// TIA Portal project "function block1" (V16)

(* hardware
DEVICE "S7-1200 station_1"  S7-1200 Station
   slot 0: "Rack_0"  S7-1200 Rack  Rack  V1.0
   slot 1: "PLC_1"  CPU 1214C DC/DC/DC  6ES7 214-1AG40-0XB0  V4.4
   slot 2: "AI 4x13BIT/AQ 2x14BIT_1"  6ES7 234-4HE32-0XB0  V2.1
   slot 101: "CP 1243-7 LTE"  CP 1243-7 LTE  6GK7 243-7KX30-0XE0  V3.2
      slot 0: "Telecontrol server"  Partner
      slot 0: "Inter-station communication"  Partner
   slot 102: "RF120C_1"  RF120C  6GT2 002-0LA00  V1.0
   slot 103: "CM 1243-5"  CM 1243-5  6GK7 243-5DX30-0XE0  V1.3
*)

// ===== PLC "PLC_1"  CPU 1214C DC/DC/DC =====

VAR_GLOBAL   // PLC tag table "Default tag table"
   "switch" AT %M0.0 : Bool;
   "out" AT %M0.1 : Bool;
   "estop" AT %M0.2 : Bool;
   "esnotification" AT %M0.3 : Bool;
   "esalarm" AT %M0.4 : Bool;
   "alarmreset" AT %M0.5 : Bool;
   "alarmsilent" AT %M0.6 : Bool;
END_VAR

DATA_BLOCK "scl_DB"   // DB1
{ S7_Optimized_Access := 'TRUE' }
VERSION : 0.1
// stored: InstanceOfName scl
"scl"
BEGIN
END_DATA_BLOCK

FUNCTION_BLOCK "scl"   // FB1, SCL
{ S7_Optimized_Access := 'TRUE' }
VERSION : 0.1
   VAR
      almset : Bool;
   END_VAR
BEGIN
   IF "estop" AND NOT #almset THEN
       "esalarm" := 1; // Statement section IF
       "esnotification" :=1;
       #almset := 1;
   END_IF;
   IF "alarmreset" AND NOT "estop" THEN
       "esalarm" := 0; // Statement section IF
       "esnotification" := 0;
       #almset := 0;
   END_IF;
   IF "alarmsilent" OR "alarmreset" AND "esnotification" THEN
       "esnotification" := 0;
   END_IF;
END_FUNCTION_BLOCK

ORGANIZATION_BLOCK "Main"   // OB1, LAD, ProgramCycle
TITLE = "Main Program Sweep (Cycle)"
{ S7_Optimized_Access := 'TRUE' }
VERSION : 0.1
   VAR_INPUT
      Initial_Call : Bool;   // Initial call of this OB
      Remanence : Bool;   // =True, if remanent data are available
   END_VAR
BEGIN

REGION Network 1
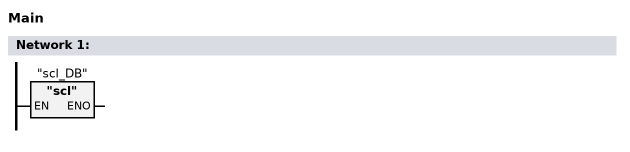
   RUNG wire#powerrail
      "scl_DB"()
   END_RUNG
   // the same network as SCL:
   "scl_DB"();   // "scl"
END_REGION
END_ORGANIZATION_BLOCK